FUNCTION_BLOCK Tabla_FIFO
VAR_INPUT 
	Dato :REAL;
END_VAR
VAR_OUTPUT
END_VAR
VAR_IN_OUT
	Tabla :ARRAY [1..10]OF REAL;
	Trigger :BOOL;
END_VAR
VAR
	posicion: INT;
END_VAR

IF trigger  THEN
	posicion:=1;
	FOR posicion:=10 TO 2 BY -1 DO
	Tabla[posicion]:=Tabla[posicion-1];
	END_FOR;
	Tabla[1]:=Dato;
	trigger:=FALSE;
END_IF

END_FUNCTION_BLOCK

(* stored: Version 1.1.0.1, ProductVersion 3.1.4024.12
   POU Tabla_FIFO: Id {1e18d4a0-ee90-4226-8a09-bcb2f67d2fe2}, SpecialFunc None *)
